Fanuc KAREL source: kf00115.KL

PROGRAM KF00115
%STACKSIZE=65535
%PRIORITY=65535
%NOLOCKGROUP
VAR
I : INTEGER
J : INTEGER
X : REAL
Y : REAL
B : BOOLEAN
C : BOOLEAN
TXT : STRING[80]
TXT2 : STRING[80]
AI : ARRAY[4] OF INTEGER
BI : ARRAY[4] OF INTEGER
P : XYZWPR
JP : JOINTPOS9
PF : POSITION
STATUS : INTEGER
-- UNRESOLVED DECLARATIONS (source type spelling not recovered)
-- V1 : TYPE_0x0013 (type_u16=0x0013)
-- V2 : TYPE_0x0013 (type_u16=0x0013)
ROUTINE FADD(P1 : INTEGER) : INTEGER FROM KF00115
ROUTINE FADD
BEGIN
-- UNRESOLVED_PC line 22 opcodes [2D 9D 52 7F] marker_code=1
-- UNRESOLVED_PC line 23 opcodes [7F] marker_code=18
END FADD
BEGIN
I=FADD(2)
END KF00115
